TEST_FINISHED();
END_METHOD

METHOD PUBLIC Check_DATE_TO_TOD_TooHigh
VAR
	value : DATE := DatatypeLimits.DATE_MAX_VALUE;
	actual : TOD;
	converted : BOOL;
END_VAR
TEST('Check_DATE_TO_TOD_TooHigh');

// @TEST-RUN
converted := TryConvert_DATE_TO_Destination(value, actual);

// @TEST-ASSERT
AssertFalse(Condition := converted, Message := 'Did not report DATE to TOD conversion was prevented');

TEST_FINISHED();
END_METHOD

METHOD PUBLIC Check_DATE_TO_TOD_Max
VAR
	value : DATE := DatatypeLimits.MAX_VALUE_OF_DATE_WHICH_CAN_BE_HELD_IN_A_TOD;
	actual : TOD;
	converted : BOOL;
	equal : BOOL;
END_VAR
TEST('Check_DATE_TO_TOD_Max');

// @TEST-RUN
converted := TryConvert_DATE_TO_Destination(value, actual);
equal := actual = DATE_TO_TOD(value);

// @TEST-ASSERT
AssertTrue(Condition := equal, Message := 'Did not convert DATE to TOD correctly');
AssertTrue(Condition := converted, Message := 'Did not report DATE to TOD conversion was successful');

TEST_FINISHED();
END_METHOD

METHOD PUBLIC Check_DATE_TO_UDINT_Min
VAR
	value : DATE := DatatypeLimits.DATE_MIN_VALUE;
	actual : UDINT;
	converted : BOOL;
	equal : BOOL;
END_VAR
TEST('Check_DATE_TO_UDINT_Min');

// @TEST-RUN
converted := TryConvert_DATE_TO_Destination(value, actual);
equal := actual = DATE_TO_UDINT(value);

// @TEST-ASSERT
AssertTrue(Condition := equal, Message := 'Did not convert DATE to UDINT correctly');
AssertTrue(Condition := converted, Message := 'Did not report DATE to UDINT conversion was successful');

TEST_FINISHED();
END_METHOD

METHOD PUBLIC Check_DATE_TO_UDINT_Max
VAR
	value : DATE := DatatypeLimits.DATE_MAX_VALUE;
	actual : UDINT;
	converted : BOOL;
	equal : BOOL;
END_VAR
TEST('Check_DATE_TO_UDINT_Max');

// @TEST-RUN
converted := TryConvert_DATE_TO_Destination(value, actual);
equal := actual = DATE_TO_UDINT(value);

// @TEST-ASSERT
AssertTrue(Condition := equal, Message := 'Did not convert DATE to UDINT correctly');
AssertTrue(Condition := converted, Message := 'Did not report DATE to UDINT conversion was successful');

TEST_FINISHED();
END_METHOD

METHOD PUBLIC Check_DATE_TO_UINT_Min
VAR
	value : DATE := DatatypeLimits.DATE_MIN_VALUE;
	actual : UINT;
	converted : BOOL;
	equal : BOOL;
END_VAR
TEST('Check_DATE_TO_UINT_Min');

// @TEST-RUN
converted := TryConvert_DATE_TO_Destination(value, actual);
equal := actual = DATE_TO_UINT(value);

// @TEST-ASSERT
AssertTrue(Condition := equal, Message := 'Did not convert DATE to UINT correctly');
AssertTrue(Condition := converted, Message := 'Did not report DATE to UINT conversion was successful');

TEST_FINISHED();
END_METHOD

METHOD PUBLIC Check_DATE_TO_UINT_TooHigh
VAR
	value : DATE := DatatypeLimits.DATE_MAX_VALUE;
	actual : UINT;
	converted : BOOL;
END_VAR
TEST('Check_DATE_TO_UINT_TooHigh');

// @TEST-RUN
converted := TryConvert_DATE_TO_Destination(value, actual);

// @TEST-ASSERT
AssertFalse(Condition := converted, Message := 'Did not report DATE to UINT conversion was prevented');

TEST_FINISHED();
END_METHOD

METHOD PUBLIC Check_DATE_TO_UINT_Max
VAR
	value : DATE := DatatypeLimits.MAX_VALUE_OF_DATE_WHICH_CAN_BE_HELD_IN_A_UINT;
	actual : UINT;
	converted : BOOL;
	equal : BOOL;
END_VAR
TEST('Check_DATE_TO_UINT_Max');

// @TEST-RUN
converted := TryConvert_DATE_TO_Destination(value, actual);
equal := actual = DATE_TO_UINT(value);

// @TEST-ASSERT
AssertTrue(Condition := equal, Message := 'Did not convert DATE to UINT correctly');
AssertTrue(Condition := converted, Message := 'Did not report DATE to UINT conversion was successful');

TEST_FINISHED();
END_METHOD

METHOD PUBLIC Check_DATE_TO_ULINT_Min
VAR
	value : DATE := DatatypeLimits.DATE_MIN_VALUE;
	actual : ULINT;
	converted : BOOL;
	equal : BOOL;
END_VAR
TEST('Check_DATE_TO_ULINT_Min');

// @TEST-RUN
converted := TryConvert_DATE_TO_Destination(value, actual);
equal := actual = DATE_TO_ULINT(value);

// @TEST-ASSERT
AssertTrue(Condition := equal, Message := 'Did not convert DATE to ULINT correctly');
AssertTrue(Condition := converted, Message := 'Did not report DATE to ULINT conversion was successful');

TEST_FINISHED();
END_METHOD

METHOD PUBLIC Check_DATE_TO_ULINT_Max
VAR
	value : DATE := DatatypeLimits.DATE_MAX_VALUE;
	actual : ULINT;
	converted : BOOL;
	equal : BOOL;
END_VAR
TEST('Check_DATE_TO_ULINT_Max');

// @TEST-RUN
converted := TryConvert_DATE_TO_Destination(value, actual);
equal := actual = DATE_TO_ULINT(value);

// @TEST-ASSERT
AssertTrue(Condition := equal, Message := 'Did not convert DATE to ULINT correctly');
AssertTrue(Condition := converted, Message := 'Did not report DATE to ULINT conversion was successful');

TEST_FINISHED();
END_METHOD

METHOD PUBLIC Check_DATE_TO_USINT_Min
VAR
	value : DATE := DatatypeLimits.DATE_MIN_VALUE;
	actual : USINT;
	converted : BOOL;
	equal : BOOL;
END_VAR
TEST('Check_DATE_TO_USINT_Min');

// @TEST-RUN
converted := TryConvert_DATE_TO_Destination(value, actual);
equal := actual = DATE_TO_USINT(value);

// @TEST-ASSERT
AssertTrue(Condition := equal, Message := 'Did not convert DATE to USINT correctly');
AssertTrue(Condition := converted, Message := 'Did not report DATE to USINT conversion was successful');

TEST_FINISHED();
END_METHOD

METHOD PUBLIC Check_DATE_TO_USINT_TooHigh
VAR
	value : DATE := DatatypeLimits.DATE_MAX_VALUE;
	actual : USINT;
	converted : BOOL;
END_VAR
TEST('Check_DATE_TO_USINT_TooHigh');

// @TEST-RUN
converted := TryConvert_DATE_TO_Destination(value, actual);

// @TEST-ASSERT
AssertFalse(Condition := converted, Message := 'Did not report DATE to USINT conversion was prevented');

TEST_FINISHED();
END_METHOD

METHOD PUBLIC Check_DATE_TO_USINT_Max
VAR
	value : DATE := DatatypeLimits.MAX_VALUE_OF_DATE_WHICH_CAN_BE_HELD_IN_A_USINT;
	actual : USINT;
	converted : BOOL;
	equal : BOOL;
END_VAR
TEST('Check_DATE_TO_USINT_Max');

// @TEST-RUN
converted := TryConvert_DATE_TO_Destination(value, actual);
equal := actual = DATE_TO_USINT(value);

// @TEST-ASSERT
AssertTrue(Condition := equal, Message := 'Did not convert DATE to USINT correctly');
AssertTrue(Condition := converted, Message := 'Did not report DATE to USINT conversion was successful');

TEST_FINISHED();
END_METHOD

METHOD PUBLIC Check_DATE_TO_WORD_Min
VAR
	value : DATE := DatatypeLimits.DATE_MIN_VALUE;
	actual : WORD;
	converted : BOOL;
	equal : BOOL;
END_VAR
TEST('Check_DATE_TO_WORD_Min');

// @TEST-RUN
converted := TryConvert_DATE_TO_Destination(value, actual);
equal := actual = DATE_TO_WORD(value);

// @TEST-ASSERT
AssertTrue(Condition := equal, Message := 'Did not convert DATE to WORD correctly');
AssertTrue(Condition := converted, Message := 'Did not report DATE to WORD conversion was successful');

TEST_FINISHED();
END_METHOD

METHOD PUBLIC Check_DATE_TO_WORD_TooHigh
VAR
	value : DATE := DatatypeLimits.DATE_MAX_VALUE;
	actual : WORD;
	converted : BOOL;
END_VAR
TEST('Check_DATE_TO_WORD_TooHigh');

// @TEST-RUN
converted := TryConvert_DATE_TO_Destination(value, actual);

// @TEST-ASSERT
AssertFalse(Condition := converted, Message := 'Did not report DATE to WORD conversion was prevented');

TEST_FINISHED();
END_METHOD

METHOD PUBLIC Check_DATE_TO_WORD_Max
VAR
	value : DATE := DatatypeLimits.MAX_VALUE_OF_DATE_WHICH_CAN_BE_HELD_IN_A_WORD;
	actual : WORD;
	converted : BOOL;
	equal : BOOL;
END_VAR
TEST('Check_DATE_TO_WORD_Max');

// @TEST-RUN
converted := TryConvert_DATE_TO_Destination(value, actual);
equal := actual = DATE_TO_WORD(value);

// @TEST-ASSERT
AssertTrue(Condition := equal, Message := 'Did not convert DATE to WORD correctly');
AssertTrue(Condition := converted, Message := 'Did not report DATE to WORD conversion was successful');

TEST_FINISHED();
END_METHOD

END_FUNCTION_BLOCK

// ---- Tests/DT_TO_TestSuite.TcPOU
FUNCTION_BLOCK PUBLIC DT_TO_TestSuite EXTENDS TcUnit.FB_TestSuite
VAR
END_VAR

Check_DT_TO_BOOL_Max();
Check_DT_TO_BOOL_Min();
Check_DT_TO_BYTE_Max();
Check_DT_TO_BYTE_Min();
Check_DT_TO_BYTE_TooHigh();
Check_DT_TO_WORD_Max();
Check_DT_TO_WORD_Min();
Check_DT_TO_WORD_TooHigh();
Check_DT_TO_DWORD_Max();
Check_DT_TO_DWORD_Min();
Check_DT_TO_LWORD_Max();
Check_DT_TO_LWORD_Min();
Check_DT_TO_SINT_Max();
Check_DT_TO_SINT_Min();
Check_DT_TO_SINT_TooHigh();
Check_DT_TO_INT_Max();
Check_DT_TO_INT_Min();
Check_DT_TO_INT_TooHigh();
Check_DT_TO_DINT_Max();
Check_DT_TO_DINT_Min();
Check_DT_TO_DINT_TooHigh();
Check_DT_TO_LINT_Max();
Check_DT_TO_LINT_Min();
Check_DT_TO_USINT_Max();
Check_DT_TO_USINT_Min();
Check_DT_TO_USINT_TooHigh();
Check_DT_TO_UINT_Max();
Check_DT_TO_UINT_Min();
Check_DT_TO_UINT_TooHigh();
Check_DT_TO_UDINT_Max();
Check_DT_TO_UDINT_Min();
Check_DT_TO_ULINT_Max();
Check_DT_TO_ULINT_Min();
Check_DT_TO_REAL_Max();
Check_DT_TO_REAL_Min();
Check_DT_TO_LREAL_Max();
Check_DT_TO_LREAL_Min();
Check_DT_TO_TIME_Max();
Check_DT_TO_TIME_Min();
Check_DT_TO_TIME_TooHigh();
Check_DT_TO_TOD_Max();
Check_DT_TO_TOD_Min();
Check_DT_TO_TOD_TooHigh();
Check_DT_TO_DATE_Max();
Check_DT_TO_DATE_Min();
Check_DT_TO_DT_Max();
Check_DT_TO_DT_Min();
Check_DT_TO_STRING_Max();
Check_DT_TO_STRING_Min();

METHOD PUBLIC Check_DT_TO_BOOL_Min
VAR
	value : DT := DatatypeLimits.DT_MIN_VALUE;
	actual : BOOL;
	converted : BOOL;
	equal : BOOL;
END_VAR
TEST('Check_DT_TO_BOOL_Min');

// @TEST-RUN
converted := TryConvert_DT_TO_Destination(value, actual);
equal := actual = DT_TO_BOOL(value);

// @TEST-ASSERT
AssertTrue(Condition := equal, Message := 'Did not convert DT to BOOL correctly');
AssertTrue(Condition := converted, Message := 'Did not report DT to BOOL conversion was successful');

TEST_FINISHED();
END_METHOD

METHOD PUBLIC Check_DT_TO_BOOL_Max
VAR
	value : DT := DatatypeLimits.DT_MAX_VALUE;
	actual : BOOL;
	converted : BOOL;
	equal : BOOL;
END_VAR
TEST('Check_DT_TO_BOOL_Max');

// @TEST-RUN
converted := TryConvert_DT_TO_Destination(value, actual);
equal := actual = DT_TO_BOOL(value);

// @TEST-ASSERT
AssertTrue(Condition := equal, Message := 'Did not convert DT to BOOL correctly');
AssertTrue(Condition := converted, Message := 'Did not report DT to BOOL conversion was successful');

TEST_FINISHED();
END_METHOD

METHOD PUBLIC Check_DT_TO_BYTE_Min
VAR
	value : DT := DatatypeLimits.DT_MIN_VALUE;
	actual : BYTE;
	converted : BOOL;
	equal : BOOL;
END_VAR
TEST('Check_DT_TO_BYTE_Min');

// @TEST-RUN
converted := TryConvert_DT_TO_Destination(value, actual);
equal := actual = DT_TO_BYTE(value);

// @TEST-ASSERT
AssertTrue(Condition := equal, Message := 'Did not convert DT to BYTE correctly');
AssertTrue(Condition := converted, Message := 'Did not report DT to BYTE conversion was successful');

TEST_FINISHED();
END_METHOD

METHOD PUBLIC Check_DT_TO_BYTE_TooHigh
VAR
	value : DT := DatatypeLimits.DT_MAX_VALUE;
	actual : BYTE;
	converted : BOOL;
END_VAR
TEST('Check_DT_TO_BYTE_TooHigh');

// @TEST-RUN
converted := TryConvert_DT_TO_Destination(value, actual);

// @TEST-ASSERT
AssertFalse(Condition := converted, Message := 'Did not report DT to BYTE conversion was prevented');

TEST_FINISHED();
END_METHOD

METHOD PUBLIC Check_DT_TO_BYTE_Max
VAR
	value : DT := DatatypeLimits.MAX_VALUE_OF_DT_WHICH_CAN_BE_HELD_IN_A_BYTE;
	actual : BYTE;
	converted : BOOL;
	equal : BOOL;
END_VAR
TEST('Check_DT_TO_BYTE_Max');

// @TEST-RUN
converted := TryConvert_DT_TO_Destination(value, actual);
equal := actual = DT_TO_BYTE(value);

// @TEST-ASSERT
AssertTrue(Condition := equal, Message := 'Did not convert DT to BYTE correctly');
AssertTrue(Condition := converted, Message := 'Did not report DT to BYTE conversion was successful');

TEST_FINISHED();
END_METHOD

METHOD PUBLIC Check_DT_TO_DATE_Min
VAR
	value : DT := DatatypeLimits.DT_MIN_VALUE;
	actual : DATE;
	converted : BOOL;
	equal : BOOL;
END_VAR
TEST('Check_DT_TO_DATE_Min');

// @TEST-RUN
converted := TryConvert_DT_TO_Destination(value, actual);
equal := actual = DT_TO_DATE(value);

// @TEST-ASSERT
AssertTrue(Condition := equal, Message := 'Did not convert DT to DATE correctly');
AssertTrue(Condition := converted, Message := 'Did not report DT to DATE conversion was successful');

TEST_FINISHED();
END_METHOD

METHOD PUBLIC Check_DT_TO_DATE_Max
VAR
	value : DT := DatatypeLimits.DT_MAX_VALUE;
	actual : DATE;
	converted : BOOL;
	equal : BOOL;
END_VAR
TEST('Check_DT_TO_DATE_Max');

// @TEST-RUN
converted := TryConvert_DT_TO_Destination(value, actual);
equal := actual = DT_TO_DATE(value);

// @TEST-ASSERT
AssertTrue(Condition := equal, Message := 'Did not convert DT to DATE correctly');
AssertTrue(Condition := converted, Message := 'Did not report DT to DATE conversion was successful');

TEST_FINISHED();
END_METHOD

METHOD PUBLIC Check_DT_TO_DINT_Min
VAR
	value : DT := DatatypeLimits.DT_MIN_VALUE;
	actual : DINT;
	converted : BOOL;
	equal : BOOL;
END_VAR
TEST('Check_DT_TO_DINT_Min');

// @TEST-RUN
converted := TryConvert_DT_TO_Destination(value, actual);
equal := actual = DT_TO_DINT(value);

// @TEST-ASSERT
AssertTrue(Condition := equal, Message := 'Did not convert DT to DINT correctly');
AssertTrue(Condition := converted, Message := 'Did not report DT to DINT conversion was successful');

TEST_FINISHED();
END_METHOD

METHOD PUBLIC Check_DT_TO_DINT_TooHigh
VAR
	value : DT := DatatypeLimits.DT_MAX_VALUE;
	actual : DINT;
	converted : BOOL;
END_VAR
TEST('Check_DT_TO_DINT_TooHigh');

// @TEST-RUN
converted := TryConvert_DT_TO_Destination(value, actual);

// @TEST-ASSERT
AssertFalse(Condition := converted, Message := 'Did not report DT to DINT conversion was prevented');

TEST_FINISHED();
END_METHOD

METHOD PUBLIC Check_DT_TO_DINT_Max
VAR
	value : DT := DatatypeLimits.MAX_VALUE_OF_DT_WHICH_CAN_BE_HELD_IN_A_DINT;
	actual : DINT;
	converted : BOOL;
	equal : BOOL;
END_VAR
TEST('Check_DT_TO_DINT_Max');

// @TEST-RUN
converted := TryConvert_DT_TO_Destination(value, actual);
equal := actual = DT_TO_DINT(value);

// @TEST-ASSERT
AssertTrue(Condition := equal, Message := 'Did not convert DT to DINT correctly');
AssertTrue(Condition := converted, Message := 'Did not report DT to DINT conversion was successful');

TEST_FINISHED();
END_METHOD

METHOD PUBLIC Check_DT_TO_DT_Min
VAR
	value : DT := DatatypeLimits.DT_MIN_VALUE;
	actual : DT;
	converted : BOOL;
	equal : BOOL;
END_VAR
TEST('Check_DT_TO_DT_Min');

// @TEST-RUN
converted := TryConvert_DT_TO_Destination(value, actual);
equal := actual = value;

// @TEST-ASSERT
AssertTrue(Condition := equal, Message := 'Did not convert DT to DT correctly');
AssertTrue(Condition := converted, Message := 'Did not report DT to DT conversion was successful');

TEST_FINISHED();
END_METHOD

METHOD PUBLIC Check_DT_TO_DT_Max
VAR
	value : DT := DatatypeLimits.DT_MAX_VALUE;
	actual : DT;
	converted : BOOL;
	equal : BOOL;
END_VAR
TEST('Check_DT_TO_DT_Max');

// @TEST-RUN
converted := TryConvert_DT_TO_Destination(value, actual);
equal := actual = value;

// @TEST-ASSERT
AssertTrue(Condition := equal, Message := 'Did not convert DT to DT correctly');
AssertTrue(Condition := converted, Message := 'Did not report DT to DT conversion was successful');

TEST_FINISHED();
END_METHOD

METHOD PUBLIC Check_DT_TO_DWORD_Min
VAR
	value : DT := DatatypeLimits.DT_MIN_VALUE;
	actual : DWORD;
	converted : BOOL;
	equal : BOOL;
END_VAR
TEST('Check_DT_TO_DWORD_Min');

// @TEST-RUN
converted := TryConvert_DT_TO_Destination(value, actual);
equal := actual = DT_TO_DWORD(value);

// @TEST-ASSERT
AssertTrue(Condition := equal, Message := 'Did not convert DT to DWORD correctly');
AssertTrue(Condition := converted, Message := 'Did not report DT to DWORD conversion was successful');

TEST_FINISHED();
END_METHOD

METHOD PUBLIC Check_DT_TO_DWORD_Max
VAR
	value : DT := DatatypeLimits.DT_MAX_VALUE;
	actual : DWORD;
	converted : BOOL;
	equal : BOOL;
END_VAR
TEST('Check_DT_TO_DWORD_Max');

// @TEST-RUN
converted := TryConvert_DT_TO_Destination(value, actual);
equal := actual = DT_TO_DWORD(value);

// @TEST-ASSERT
AssertTrue(Condition := equal, Message := 'Did not convert DT to DWORD correctly');
AssertTrue(Condition := converted, Message := 'Did not report DT to DWORD conversion was successful');

TEST_FINISHED();
END_METHOD

METHOD PUBLIC Check_DT_TO_INT_Min
VAR
	value : DT := DatatypeLimits.DT_MIN_VALUE;
	actual : INT;
	converted : BOOL;
	equal : BOOL;
END_VAR
TEST('Check_DT_TO_INT_Min');

// @TEST-RUN
converted := TryConvert_DT_TO_Destination(value, actual);
equal := actual = DT_TO_INT(value);

// @TEST-ASSERT
AssertTrue(Condition := equal, Message := 'Did not convert DT to INT correctly');
AssertTrue(Condition := converted, Message := 'Did not report DT to INT conversion was successful');

TEST_FINISHED();
END_METHOD

METHOD PUBLIC Check_DT_TO_INT_TooHigh
VAR
	value : DT := DatatypeLimits.DT_MAX_VALUE;
	actual : INT;
	converted : BOOL;
END_VAR
TEST('Check_DT_TO_INT_TooHigh');

// @TEST-RUN
converted := TryConvert_DT_TO_Destination(value, actual);

// @TEST-ASSERT
AssertFalse(Condition := converted, Message := 'Did not report DT to INT conversion was prevented');

TEST_FINISHED();
END_METHOD

METHOD PUBLIC Check_DT_TO_INT_Max
VAR
	value : DT := DatatypeLimits.MAX_VALUE_OF_DT_WHICH_CAN_BE_HELD_IN_A_INT;
	actual : INT;
	converted : BOOL;
	equal : BOOL;
END_VAR
TEST('Check_DT_TO_INT_Max');

// @TEST-RUN
converted := TryConvert_DT_TO_Destination(value, actual);
equal := actual = DT_TO_INT(value);

// @TEST-ASSERT
AssertTrue(Condition := equal, Message := 'Did not convert DT to INT correctly');
AssertTrue(Condition := converted, Message := 'Did not report DT to INT conversion was successful');

TEST_FINISHED();
END_METHOD

METHOD PUBLIC Check_DT_TO_LINT_Min
VAR
	value : DT := DatatypeLimits.DT_MIN_VALUE;
	actual : LINT;
	converted : BOOL;
	equal : BOOL;
END_VAR
TEST('Check_DT_TO_LINT_Min');

// @TEST-RUN
converted := TryConvert_DT_TO_Destination(value, actual);
equal := actual = DT_TO_LINT(value);

// @TEST-ASSERT
AssertTrue(Condition := equal, Message := 'Did not convert DT to LINT correctly');
AssertTrue(Condition := converted, Message := 'Did not report DT to LINT conversion was successful');

TEST_FINISHED();
END_METHOD

METHOD PUBLIC Check_DT_TO_LINT_Max
VAR
	value : DT := DatatypeLimits.DT_MAX_VALUE;
	actual : LINT;
	converted : BOOL;
	equal : BOOL;
END_VAR
TEST('Check_DT_TO_LINT_Max');

// @TEST-RUN
converted := TryConvert_DT_TO_Destination(value, actual);
equal := actual = DT_TO_LINT(value);

// @TEST-ASSERT
AssertTrue(Condition := equal, Message := 'Did not convert DT to LINT correctly');
AssertTrue(Condition := converted, Message := 'Did not report DT to LINT conversion was successful');

TEST_FINISHED();
END_METHOD

METHOD PUBLIC Check_DT_TO_LREAL_Min
VAR
	value : DT := DatatypeLimits.DT_MIN_VALUE;
	actual : LREAL;
	converted : BOOL;
	equal : BOOL;
END_VAR
TEST('Check_DT_TO_LREAL_Min');

// @TEST-RUN
converted := TryConvert_DT_TO_Destination(value, actual);
equal := actual = DT_TO_LREAL(value);

// @TEST-ASSERT
AssertTrue(Condition := equal, Message := 'Did not convert DT to LREAL correctly');
AssertTrue(Condition := converted, Message := 'Did not report DT to LREAL conversion was successful');

TEST_FINISHED();
END_METHOD

METHOD PUBLIC Check_DT_TO_LREAL_Max
VAR
	value : DT := DatatypeLimits.DT_MAX_VALUE;
	actual : LREAL;
	converted : BOOL;
	equal : BOOL;
END_VAR
TEST('Check_DT_TO_LREAL_Max');

// @TEST-RUN
converted := TryConvert_DT_TO_Destination(value, actual);
equal := actual = DT_TO_LREAL(value);

// @TEST-ASSERT
AssertTrue(Condition := equal, Message := 'Did not convert DT to LREAL correctly');
AssertTrue(Condition := converted, Message := 'Did not report DT to LREAL conversion was successful');

TEST_FINISHED();
END_METHOD

METHOD PUBLIC Check_DT_TO_LWORD_Min
VAR
	value : DT := DatatypeLimits.DT_MIN_VALUE;
	actual : LWORD;
	converted : BOOL;
	equal : BOOL;
END_VAR
TEST('Check_DT_TO_LWORD_Min');

// @TEST-RUN
converted := TryConvert_DT_TO_Destination(value, actual);
equal := actual = DT_TO_LWORD(value);

// @TEST-ASSERT
AssertTrue(Condition := equal, Message := 'Did not convert DT to LWORD correctly');
AssertTrue(Condition := converted, Message := 'Did not report DT to LWORD conversion was successful');

TEST_FINISHED();
END_METHOD

METHOD PUBLIC Check_DT_TO_LWORD_Max
VAR
	value : DT := DatatypeLimits.DT_MAX_VALUE;
	actual : LWORD;
	converted : BOOL;
	equal : BOOL;
END_VAR
TEST('Check_DT_TO_LWORD_Max');

// @TEST-RUN
converted := TryConvert_DT_TO_Destination(value, actual);
equal := actual = DT_TO_LWORD(value);

// @TEST-ASSERT
AssertTrue(Condition := equal, Message := 'Did not convert DT to LWORD correctly');
AssertTrue(Condition := converted, Message := 'Did not report DT to LWORD conversion was successful');

TEST_FINISHED();
END_METHOD

METHOD PUBLIC Check_DT_TO_REAL_Min
VAR
	value : DT := DatatypeLimits.DT_MIN_VALUE;
	actual : REAL;
	converted : BOOL;
	equal : BOOL;
END_VAR
TEST('Check_DT_TO_REAL_Min');

// @TEST-RUN
converted := TryConvert_DT_TO_Destination(value, actual);
equal := actual = DT_TO_REAL(value);

// @TEST-ASSERT
AssertTrue(Condition := equal, Message := 'Did not convert DT to REAL correctly');
AssertTrue(Condition := converted, Message := 'Did not report DT to REAL conversion was successful');

TEST_FINISHED();
END_METHOD

METHOD PUBLIC Check_DT_TO_REAL_Max
VAR
	value : DT := DatatypeLimits.DT_MAX_VALUE;
	actual : REAL;
	converted : BOOL;
	equal : BOOL;
END_VAR
TEST('Check_DT_TO_REAL_Max');

// @TEST-RUN
converted := TryConvert_DT_TO_Destination(value, actual);
equal := actual = DT_TO_REAL(value);

// @TEST-ASSERT
AssertTrue(Condition := equal, Message := 'Did not convert DT to REAL correctly');
AssertTrue(Condition := converted, Message := 'Did not report DT to REAL conversion was successful');

TEST_FINISHED();
END_METHOD

METHOD PUBLIC Check_DT_TO_SINT_Min
VAR
	value : DT := DatatypeLimits.DT_MIN_VALUE;
	actual : SINT;
	converted : BOOL;
	equal : BOOL;
END_VAR
TEST('Check_DT_TO_SINT_Min');

// @TEST-RUN
converted := TryConvert_DT_TO_Destination(value, actual);
equal := actual = DT_TO_SINT(value);

// @TEST-ASSERT
AssertTrue(Condition := equal, Message := 'Did not convert DT to SINT correctly');
AssertTrue(Condition := converted, Message := 'Did not report DT to SINT conversion was successful');

TEST_FINISHED();
END_METHOD

METHOD PUBLIC Check_DT_TO_SINT_TooHigh
VAR
	value : DT := DatatypeLimits.DT_MAX_VALUE;
	actual : SINT;
	converted : BOOL;
END_VAR
TEST('Check_DT_TO_SINT_TooHigh');

// @TEST-RUN
converted := TryConvert_DT_TO_Destination(value, actual);

// @TEST-ASSERT
AssertFalse(Condition := converted, Message := 'Did not report DT to SINT conversion was prevented');

TEST_FINISHED();
END_METHOD

METHOD PUBLIC Check_DT_TO_SINT_Max
VAR
	value : DT := DatatypeLimits.MAX_VALUE_OF_DT_WHICH_CAN_BE_HELD_IN_A_SINT;
	actual : SINT;
	converted : BOOL;
	equal : BOOL;
END_VAR
TEST('Check_DT_TO_SINT_Max');

// @TEST-RUN
converted := TryConvert_DT_TO_Destination(value, actual);
equal := actual = DT_TO_SINT(value);

// @TEST-ASSERT
AssertTrue(Condition := equal, Message := 'Did not convert DT to SINT correctly');
AssertTrue(Condition := converted, Message := 'Did not report DT to SINT conversion was successful');

TEST_FINISHED();
END_METHOD

METHOD PUBLIC Check_DT_TO_STRING_Min
VAR
	value : DT := DatatypeLimits.DT_MIN_VALUE;
	actual : STRING;
	converted : BOOL;
	equal : BOOL;
END_VAR
TEST('Check_DT_TO_STRING_Min');

// @TEST-RUN
converted := TryConvert_DT_TO_Destination(value, actual);
equal := actual = DT_TO_STRING(value);

// @TEST-ASSERT
AssertTrue(Condition := equal, Message := 'Did not convert DT to STRING correctly');
AssertTrue(Condition := converted, Message := 'Did not report DT to STRING conversion was successful');

TEST_FINISHED();
END_METHOD

METHOD PUBLIC Check_DT_TO_STRING_Max
VAR
	value : DT := DatatypeLimits.DT_MAX_VALUE;
	actual : STRING;
	converted : BOOL;
	equal : BOOL;
END_VAR
TEST('Check_DT_TO_STRING_Max');

// @TEST-RUN
converted := TryConvert_DT_TO_Destination(value, actual);
equal := actual = DT_TO_STRING(value);

// @TEST-ASSERT
AssertTrue(Condition := equal, Message := 'Did not convert DT to STRING correctly');
AssertTrue(Condition := converted, Message := 'Did not report DT to STRING conversion was successful');

TEST_FINISHED();
END_METHOD

METHOD PUBLIC Check_DT_TO_TIME_Min
VAR
	value : DT := DatatypeLimits.DT_MIN_VALUE;
	actual : TIME;
	converted : BOOL;
	equal : BOOL;
END_VAR
TEST('Check_DT_TO_TIME_Min');

// @TEST-RUN
converted := TryConvert_DT_TO_Destination(value, actual);
equal := actual = DT_TO_TIME(value);

// @TEST-ASSERT
AssertTrue(Condition := equal, Message := 'Did not convert DT to TIME correctly');
AssertTrue(Condition := converted, Message := 'Did not report DT to TIME conversion was successful');

TEST_FINISHED();
END_METHOD

METHOD PUBLIC Check_DT_TO_TIME_TooHigh
VAR
	value : DT := DatatypeLimits.DT_MAX_VALUE;
	actual : TIME;
	converted : BOOL;
END_VAR
TEST('Check_DT_TO_TIME_TooHigh');

// @TEST-RUN
converted := TryConvert_DT_TO_Destination(value, actual);

// @TEST-ASSERT
AssertFalse(Condition := converted, Message := 'Did not report DT to TIME conversion was prevented');

TEST_FINISHED();
END_METHOD

METHOD PUBLIC Check_DT_TO_TIME_Max
VAR
	value : DT := DatatypeLimits.MAX_VALUE_OF_DT_WHICH_CAN_BE_HELD_IN_A_TIME;
	actual : TIME;
	converted : BOOL;
	equal : BOOL;
END_VAR
TEST('Check_DT_TO_TIME_Max');

// @TEST-RUN
converted := TryConvert_DT_TO_Destination(value, actual);
equal := actual = DT_TO_TIME(value);

// @TEST-ASSERT
AssertTrue(Condition := equal, Message := 'Did not convert DT to TIME correctly');
AssertTrue(Condition := converted, Message := 'Did not report DT to TIME conversion was successful');

TEST_FINISHED();
END_METHOD

METHOD PUBLIC Check_DT_TO_TOD_Min
VAR
	value : DT := DatatypeLimits.DT_MIN_VALUE;
	actual : TOD;
	converted : BOOL;
	equal : BOOL;
END_VAR
TEST('Check_DT_TO_TOD_Min');

// @TEST-RUN
converted := TryConvert_DT_TO_Destination(value, actual);
equal := actual = DT_TO_TOD(value);

// @TEST-ASSERT
AssertTrue(Condition := equal, Message := 'Did not convert DT to TOD correctly');
AssertTrue(Condition := converted, Message := 'Did not report DT to TOD conversion was successful');

TEST_FINISHED();
END_METHOD

METHOD PUBLIC Check_DT_TO_TOD_TooHigh
VAR
	value : DT := DatatypeLimits.DT_MAX_VALUE;
	actual : TOD;
	converted : BOOL;
END_VAR
TEST('Check_DT_TO_TOD_TooHigh');

// @TEST-RUN
converted := TryConvert_DT_TO_Destination(value, actual);

// @TEST-ASSERT
AssertFalse(Condition := converted, Message := 'Did not report DT to TOD conversion was prevented');

TEST_FINISHED();
END_METHOD

METHOD PUBLIC Check_DT_TO_TOD_Max
VAR
	value : DT := DatatypeLimits.MAX_VALUE_OF_DT_WHICH_CAN_BE_HELD_IN_A_TOD;
	actual : TOD;
	converted : BOOL;
	equal : BOOL;
END_VAR
TEST('Check_DT_TO_TOD_Max');

// @TEST-RUN
converted := TryConvert_DT_TO_Destination(value, actual);
equal := actual = DT_TO_TOD(value);

// @TEST-ASSERT
AssertTrue(Condition := equal, Message := 'Did not convert DT to TOD correctly');
AssertTrue(Condition := converted, Message := 'Did not report DT to TOD conversion was successful');

TEST_FINISHED();
END_METHOD

METHOD PUBLIC Check_DT_TO_UDINT_Min
VAR
	value : DT := DatatypeLimits.DT_MIN_VALUE;
	actual : UDINT;
	converted : BOOL;
	equal : BOOL;
END_VAR
TEST('Check_DT_TO_UDINT_Min');

// @TEST-RUN
converted := TryConvert_DT_TO_Destination(value, actual);
equal := actual = DT_TO_UDINT(value);

// @TEST-ASSERT
AssertTrue(Condition := equal, Message := 'Did not convert DT to UDINT correctly');
AssertTrue(Condition := converted, Message := 'Did not report DT to UDINT conversion was successful');

TEST_FINISHED();
END_METHOD

METHOD PUBLIC Check_DT_TO_UDINT_Max
VAR
	value : DT := DatatypeLimits.DT_MAX_VALUE;
	actual : UDINT;
	converted : BOOL;
	equal : BOOL;
END_VAR
TEST('Check_DT_TO_UDINT_Max');

// @TEST-RUN
converted := TryConvert_DT_TO_Destination(value, actual);
equal := actual = DT_TO_UDINT(value);

// @TEST-ASSERT
AssertTrue(Condition := equal, Message := 'Did not convert DT to UDINT correctly');
AssertTrue(Condition := converted, Message := 'Did not report DT to UDINT conversion was successful');

TEST_FINISHED();
END_METHOD

METHOD PUBLIC Check_DT_TO_UINT_Min
VAR
	value : DT := DatatypeLimits.DT_MIN_VALUE;
	actual : UINT;
	converted : BOOL;
	equal : BOOL;
END_VAR
TEST('Check_DT_TO_UINT_Min');

// @TEST-RUN
converted := TryConvert_DT_TO_Destination(value, actual);
equal := actual = DT_TO_UINT(value);

// @TEST-ASSERT
AssertTrue(Condition := equal, Message := 'Did not convert DT to UINT correctly');
AssertTrue(Condition := converted, Message := 'Did not report DT to UINT conversion was successful');

TEST_FINISHED();
END_METHOD

METHOD PUBLIC Check_DT_TO_UINT_TooHigh
VAR
	value : DT := DatatypeLimits.DT_MAX_VALUE;
	actual : UINT;
	converted : BOOL;
END_VAR
TEST('Check_DT_TO_UINT_TooHigh');

// @TEST-RUN
converted := TryConvert_DT_TO_Destination(value, actual);

// @TEST-ASSERT
AssertFalse(Condition := converted, Message := 'Did not report DT to UINT conversion was prevented');

TEST_FINISHED();
END_METHOD

METHOD PUBLIC Check_DT_TO_UINT_Max
VAR
	value : DT := DatatypeLimits.MAX_VALUE_OF_DT_WHICH_CAN_BE_HELD_IN_A_UINT;
	actual : UINT;
	converted : BOOL;
	equal : BOOL;
END_VAR
TEST('Check_DT_TO_UINT_Max');

// @TEST-RUN
converted := TryConvert_DT_TO_Destination(value, actual);
equal := actual = DT_TO_UINT(value);

// @TEST-ASSERT
AssertTrue(Condition := equal, Message := 'Did not convert DT to UINT correctly');
AssertTrue(Condition := converted, Message := 'Did not report DT to UINT conversion was successful');

TEST_FINISHED();
END_METHOD

METHOD PUBLIC Check_DT_TO_ULINT_Min
VAR
	value : DT := DatatypeLimits.DT_MIN_VALUE;
	actual : ULINT;
	converted : BOOL;
	equal : BOOL;
END_VAR
TEST('Check_DT_TO_ULINT_Min');

// @TEST-RUN
converted := TryConvert_DT_TO_Destination(value, actual);
equal := actual = DT_TO_ULINT(value);

// @TEST-ASSERT
AssertTrue(Condition := equal, Message := 'Did not convert DT to ULINT correctly');
AssertTrue(Condition := converted, Message := 'Did not report DT to ULINT conversion was successful');

TEST_FINISHED();
END_METHOD

METHOD PUBLIC Check_DT_TO_ULINT_Max
VAR
	value : DT := DatatypeLimits.DT_MAX_VALUE;
	actual : ULINT;
	converted : BOOL;
	equal : BOOL;
END_VAR
TEST('Check_DT_TO_ULINT_Max');

// @TEST-RUN
converted := TryConvert_DT_TO_Destination(value, actual);
equal := actual = DT_TO_ULINT(value);

// @TEST-ASSERT
AssertTrue(Condition := equal, Message := 'Did not convert DT to ULINT correctly');
AssertTrue(Condition := converted, Message := 'Did not report DT to ULINT conversion was successful');

TEST_FINISHED();
END_METHOD

METHOD PUBLIC Check_DT_TO_USINT_Min
VAR
	value : DT := DatatypeLimits.DT_MIN_VALUE;
	actual : USINT;
	converted : BOOL;
	equal : BOOL;
END_VAR
TEST('Check_DT_TO_USINT_Min');

// @TEST-RUN
converted := TryConvert_DT_TO_Destination(value, actual);
equal := actual = DT_TO_USINT(value);

// @TEST-ASSERT
AssertTrue(Condition := equal, Message := 'Did not convert DT to USINT correctly');
AssertTrue(Condition := converted, Message := 'Did not report DT to USINT conversion was successful');

TEST_FINISHED();
END_METHOD

METHOD PUBLIC Check_DT_TO_USINT_TooHigh
VAR
	value : DT := DatatypeLimits.DT_MAX_VALUE;
	actual : USINT;
	converted : BOOL;
END_VAR
TEST('Check_DT_TO_USINT_TooHigh');

// @TEST-RUN
converted := TryConvert_DT_TO_Destination(value, actual);

// @TEST-ASSERT
AssertFalse(Condition := converted, Message := 'Did not report DT to USINT conversion was prevented');

TEST_FINISHED();
END_METHOD

METHOD PUBLIC Check_DT_TO_USINT_Max
VAR
	value : DT := DatatypeLimits.MAX_VALUE_OF_DT_WHICH_CAN_BE_HELD_IN_A_USINT;
	actual : USINT;
	converted : BOOL;
	equal : BOOL;
END_VAR
TEST('Check_DT_TO_USINT_Max');

// @TEST-RUN
converted := TryConvert_DT_TO_Destination(value, actual);
equal := actual = DT_TO_USINT(value);

// @TEST-ASSERT
AssertTrue(Condition := equal, Message := 'Did not convert DT to USINT correctly');
AssertTrue(Condition := converted, Message := 'Did not report DT to USINT conversion was successful');

TEST_FINISHED();
END_METHOD

METHOD PUBLIC Check_DT_TO_WORD_Min
VAR
	value : DT := DatatypeLimits.DT_MIN_VALUE;
	actual : WORD;
	converted : BOOL;
	equal : BOOL;
END_VAR
TEST('Check_DT_TO_WORD_Min');

// @TEST-RUN
converted := TryConvert_DT_TO_Destination(value, actual);
equal := actual = DT_TO_WORD(value);

// @TEST-ASSERT
AssertTrue(Condition := equal, Message := 'Did not convert DT to WORD correctly');
AssertTrue(Condition := converted, Message := 'Did not report DT to WORD conversion was successful');

TEST_FINISHED();
END_METHOD

METHOD PUBLIC Check_DT_TO_WORD_TooHigh
VAR
	value : DT := DatatypeLimits.DT_MAX_VALUE;
	actual : WORD;
	converted : BOOL;
END_VAR
TEST('Check_DT_TO_WORD_TooHigh');

// @TEST-RUN
converted := TryConvert_DT_TO_Destination(value, actual);

// @TEST-ASSERT
AssertFalse(Condition := converted, Message := 'Did not report DT to WORD conversion was prevented');

TEST_FINISHED();
END_METHOD

METHOD PUBLIC Check_DT_TO_WORD_Max
VAR
	value : DT := DatatypeLimits.MAX_VALUE_OF_DT_WHICH_CAN_BE_HELD_IN_A_WORD;
	actual : WORD;
	converted : BOOL;
	equal : BOOL;
END_VAR
TEST('Check_DT_TO_WORD_Max');

// @TEST-RUN
converted := TryConvert_DT_TO_Destination(value, actual);
equal := actual = DT_TO_WORD(value);

// @TEST-ASSERT
AssertTrue(Condition := equal, Message := 'Did not convert DT to WORD correctly');
AssertTrue(Condition := converted, Message := 'Did not report DT to WORD conversion was successful');

TEST_FINISHED();
END_METHOD

END_FUNCTION_BLOCK

// ---- Tests/STRING_TO_TestSuite.TcPOU
FUNCTION_BLOCK PUBLIC STRING_TO_TestSuite EXTENDS TcUnit.FB_TestSuite
VAR
END_VAR

Check_STRING_TO_BOOL_Valid();
Check_STRING_TO_BYTE_Valid();
Check_STRING_TO_BYTE_Invalid();
Check_STRING_TO_WORD_Valid();
Check_STRING_TO_WORD_Invalid();
Check_STRING_TO_DWORD_Valid();
Check_STRING_TO_DWORD_Invalid();
Check_STRING_TO_LWORD_Valid();
Check_STRING_TO_LWORD_Invalid();
Check_STRING_TO_SINT_Valid();
Check_STRING_TO_SINT_Invalid();
Check_STRING_TO_INT_Valid();
Check_STRING_TO_INT_Invalid();
Check_STRING_TO_DINT_Valid();
Check_STRING_TO_DINT_Invalid();
Check_STRING_TO_LINT_Valid();
Check_STRING_TO_LINT_Invalid();
Check_STRING_TO_USINT_Valid();
Check_STRING_TO_USINT_Invalid();
Check_STRING_TO_UINT_Valid();
Check_STRING_TO_UINT_Invalid();
Check_STRING_TO_UDINT_Valid();
Check_STRING_TO_UDINT_Invalid();
Check_STRING_TO_ULINT_Valid();
Check_STRING_TO_ULINT_Invalid();
Check_STRING_TO_REAL_Valid();
Check_STRING_TO_REAL_Invalid();
Check_STRING_TO_LREAL_Valid();
Check_STRING_TO_LREAL_Invalid();
Check_STRING_TO_TIME_Valid();
Check_STRING_TO_TIME_Invalid();
Check_STRING_TO_TOD_Valid();
Check_STRING_TO_TOD_Invalid();
Check_STRING_TO_DATE_Valid();
Check_STRING_TO_DATE_Invalid();
Check_STRING_TO_DT_Valid();
Check_STRING_TO_DT_Invalid();
Check_STRING_TO_STRING_Valid();

METHOD PUBLIC Check_STRING_TO_BOOL_Valid
VAR
	value : STRING := BOOL_TO_STRING(DatatypeLimits.BOOL_MAX_VALUE);
	actual : BOOL;
	converted : BOOL;
	equal : BOOL;
END_VAR
TEST('Check_STRING_TO_BOOL_Valid');

// @TEST-RUN
converted := TryConvert_STRING_TO_Destination(value, actual);
equal := actual = STRING_TO_BOOL(value);

// @TEST-ASSERT
AssertTrue(Condition := equal, Message := 'Did not convert STRING to BOOL correctly');
AssertTrue(Condition := converted, Message := 'Did not report STRING to BOOL conversion was successful');

TEST_FINISHED();
END_METHOD

METHOD PUBLIC Check_STRING_TO_BYTE_Invalid
VAR
	value : STRING := 'hello';
	actual : BYTE;
	converted : BOOL;
END_VAR
TEST('Check_STRING_TO_BYTE_Invalid');

// @TEST-RUN
converted := TryConvert_STRING_TO_Destination(value, actual);

// @TEST-ASSERT
AssertFalse(Condition := converted, Message := 'Did not report STRING to BYTE conversion was prevented');

TEST_FINISHED();
END_METHOD

METHOD PUBLIC Check_STRING_TO_BYTE_Valid
VAR
	value : STRING := BYTE_TO_STRING(DatatypeLimits.BYTE_MAX_VALUE);
	actual : BYTE;
	converted : BOOL;
	equal : BOOL;
END_VAR
TEST('Check_STRING_TO_BYTE_Valid');

// @TEST-RUN
converted := TryConvert_STRING_TO_Destination(value, actual);
equal := actual = STRING_TO_BYTE(value);

// @TEST-ASSERT
AssertTrue(Condition := equal, Message := 'Did not convert STRING to BYTE correctly');
AssertTrue(Condition := converted, Message := 'Did not report STRING to BYTE conversion was successful');

TEST_FINISHED();
END_METHOD

METHOD PUBLIC Check_STRING_TO_DATE_Invalid
VAR
	value : STRING := 'hello';
	actual : DATE;
	converted : BOOL;
END_VAR
TEST('Check_STRING_TO_DATE_Invalid');

// @TEST-RUN
converted := TryConvert_STRING_TO_Destination(value, actual);

// @TEST-ASSERT
AssertFalse(Condition := converted, Message := 'Did not report STRING to DATE conversion was prevented');

TEST_FINISHED();
END_METHOD

METHOD PUBLIC Check_STRING_TO_DATE_Valid
VAR
	value : STRING := DATE_TO_STRING(DatatypeLimits.DATE_MAX_VALUE);
	actual : DATE;
	converted : BOOL;
	equal : BOOL;
END_VAR
TEST('Check_STRING_TO_DATE_Valid');

// @TEST-RUN
converted := TryConvert_STRING_TO_Destination(value, actual);
equal := actual = STRING_TO_DATE(value);

// @TEST-ASSERT
AssertTrue(Condition := equal, Message := 'Did not convert STRING to DATE correctly');
AssertTrue(Condition := converted, Message := 'Did not report STRING to DATE conversion was successful');

TEST_FINISHED();
END_METHOD

METHOD PUBLIC Check_STRING_TO_DINT_Invalid
VAR
	value : STRING := 'hello';
	actual : DINT;
	converted : BOOL;
END_VAR
TEST('Check_STRING_TO_DINT_Invalid');

// @TEST-RUN
converted := TryConvert_STRING_TO_Destination(value, actual);

// @TEST-ASSERT
AssertFalse(Condition := converted, Message := 'Did not report STRING to DINT conversion was prevented');

TEST_FINISHED();
END_METHOD

METHOD PUBLIC Check_STRING_TO_DINT_Valid
VAR
	value : STRING := DINT_TO_STRING(DatatypeLimits.DINT_MAX_VALUE);
	actual : DINT;
	converted : BOOL;
	equal : BOOL;
END_VAR
TEST('Check_STRING_TO_DINT_Valid');

// @TEST-RUN
converted := TryConvert_STRING_TO_Destination(value, actual);
equal := actual = STRING_TO_DINT(value);

// @TEST-ASSERT
AssertTrue(Condition := equal, Message := 'Did not convert STRING to DINT correctly');
AssertTrue(Condition := converted, Message := 'Did not report STRING to DINT conversion was successful');

TEST_FINISHED();
END_METHOD

METHOD PUBLIC Check_STRING_TO_DT_Invalid
VAR
	value : STRING := 'hello';
	actual : DT;
	converted : BOOL;
END_VAR
TEST('Check_STRING_TO_DT_Invalid');

// @TEST-RUN
converted := TryConvert_STRING_TO_Destination(value, actual);

// @TEST-ASSERT
AssertFalse(Condition := converted, Message := 'Did not report STRING to DT conversion was prevented');

TEST_FINISHED();
END_METHOD

METHOD PUBLIC Check_STRING_TO_DT_Valid
VAR
	value : STRING := DT_TO_STRING(DatatypeLimits.DT_MAX_VALUE);
	actual : DT;
	converted : BOOL;
	equal : BOOL;
END_VAR
TEST('Check_STRING_TO_DT_Valid');

// @TEST-RUN
converted := TryConvert_STRING_TO_Destination(value, actual);
equal := actual = STRING_TO_DT(value);

// @TEST-ASSERT
AssertTrue(Condition := equal, Message := 'Did not convert STRING to DT correctly');
AssertTrue(Condition := converted, Message := 'Did not report STRING to DT conversion was successful');

TEST_FINISHED();
END_METHOD

METHOD PUBLIC Check_STRING_TO_DWORD_Invalid
VAR
	value : STRING := 'hello';
	actual : DWORD;
	converted : BOOL;
END_VAR
TEST('Check_STRING_TO_DWORD_Invalid');

// @TEST-RUN
converted := TryConvert_STRING_TO_Destination(value, actual);

// @TEST-ASSERT
AssertFalse(Condition := converted, Message := 'Did not report STRING to DWORD conversion was prevented');

TEST_FINISHED();
END_METHOD

METHOD PUBLIC Check_STRING_TO_DWORD_Valid
VAR
	value : STRING := DWORD_TO_STRING(DatatypeLimits.DWORD_MAX_VALUE);
	actual : DWORD;
	converted : BOOL;
	equal : BOOL;
END_VAR
TEST('Check_STRING_TO_DWORD_Valid');

// @TEST-RUN
converted := TryConvert_STRING_TO_Destination(value, actual);
equal := actual = STRING_TO_DWORD(value);

// @TEST-ASSERT
AssertTrue(Condition := equal, Message := 'Did not convert STRING to DWORD correctly');
AssertTrue(Condition := converted, Message := 'Did not report STRING to DWORD conversion was successful');

TEST_FINISHED();
END_METHOD

METHOD PUBLIC Check_STRING_TO_INT_Invalid
VAR
	value : STRING := 'hello';
	actual : INT;
	converted : BOOL;
END_VAR
TEST('Check_STRING_TO_INT_Invalid');

// @TEST-RUN
converted := TryConvert_STRING_TO_Destination(value, actual);

// @TEST-ASSERT
AssertFalse(Condition := converted, Message := 'Did not report STRING to INT conversion was prevented');

TEST_FINISHED();
END_METHOD

METHOD PUBLIC Check_STRING_TO_INT_Valid
VAR
	value : STRING := INT_TO_STRING(DatatypeLimits.INT_MAX_VALUE);
	actual : INT;
	converted : BOOL;
	equal : BOOL;
END_VAR
TEST('Check_STRING_TO_INT_Valid');

// @TEST-RUN
converted := TryConvert_STRING_TO_Destination(value, actual);
equal := actual = STRING_TO_INT(value);

// @TEST-ASSERT
AssertTrue(Condition := equal, Message := 'Did not convert STRING to INT correctly');
AssertTrue(Condition := converted, Message := 'Did not report STRING to INT conversion was successful');

TEST_FINISHED();
END_METHOD

METHOD PUBLIC Check_STRING_TO_LINT_Invalid
VAR
	value : STRING := 'hello';
	actual : LINT;
	converted : BOOL;
END_VAR
TEST('Check_STRING_TO_LINT_Invalid');

// @TEST-RUN
converted := TryConvert_STRING_TO_Destination(value, actual);

// @TEST-ASSERT
AssertFalse(Condition := converted, Message := 'Did not report STRING to LINT conversion was prevented');

TEST_FINISHED();
END_METHOD

METHOD PUBLIC Check_STRING_TO_LINT_Valid
VAR
	value : STRING := LINT_TO_STRING(DatatypeLimits.LINT_MAX_VALUE);
	actual : LINT;
	converted : BOOL;
	equal : BOOL;
END_VAR
TEST('Check_STRING_TO_LINT_Valid');

// @TEST-RUN
converted := TryConvert_STRING_TO_Destination(value, actual);
equal := actual = STRING_TO_LINT(value);

// @TEST-ASSERT
AssertTrue(Condition := equal, Message := 'Did not convert STRING to LINT correctly');
AssertTrue(Condition := converted, Message := 'Did not report STRING to LINT conversion was successful');

TEST_FINISHED();
END_METHOD

METHOD PUBLIC Check_STRING_TO_LREAL_Invalid
VAR
	value : STRING := 'hello';
	actual : LREAL;
	converted : BOOL;
END_VAR
TEST('Check_STRING_TO_LREAL_Invalid');

// @TEST-RUN
converted := TryConvert_STRING_TO_Destination(value, actual);

// @TEST-ASSERT
AssertFalse(Condition := converted, Message := 'Did not report STRING to LREAL conversion was prevented');

TEST_FINISHED();
END_METHOD

METHOD PUBLIC Check_STRING_TO_LREAL_Valid
VAR
	value : STRING := LREAL_TO_STRING(DatatypeLimits.MAX_VALUE_OF_LREAL_WHICH_CAN_BE_HELD_IN_A_STRING);
	actual : LREAL;
	converted : BOOL;
	equal : BOOL;
END_VAR
TEST('Check_STRING_TO_LREAL_Valid');

// @TEST-RUN
converted := TryConvert_STRING_TO_Destination(value, actual);
equal := actual = STRING_TO_LREAL(value);

// @TEST-ASSERT
AssertTrue(Condition := equal, Message := 'Did not convert STRING to LREAL correctly');
AssertTrue(Condition := converted, Message := 'Did not report STRING to LREAL conversion was successful');

TEST_FINISHED();
END_METHOD

METHOD PUBLIC Check_STRING_TO_LWORD_Invalid
VAR
	value : STRING := 'hello';
	actual : LWORD;
	converted : BOOL;
END_VAR
TEST('Check_STRING_TO_LWORD_Invalid');

// @TEST-RUN
converted := TryConvert_STRING_TO_Destination(value, actual);

// @TEST-ASSERT
AssertFalse(Condition := converted, Message := 'Did not report STRING to LWORD conversion was prevented');

TEST_FINISHED();
END_METHOD

METHOD PUBLIC Check_STRING_TO_LWORD_Valid
VAR
	value : STRING := LWORD_TO_STRING(DatatypeLimits.LWORD_MAX_VALUE);
	actual : LWORD;
	converted : BOOL;
	equal : BOOL;
END_VAR
TEST('Check_STRING_TO_LWORD_Valid');

// @TEST-RUN
converted := TryConvert_STRING_TO_Destination(value, actual);
equal := actual = STRING_TO_LWORD(value);

// @TEST-ASSERT
AssertTrue(Condition := equal, Message := 'Did not convert STRING to LWORD correctly');
AssertTrue(Condition := converted, Message := 'Did not report STRING to LWORD conversion was successful');

TEST_FINISHED();
END_METHOD

METHOD PUBLIC Check_STRING_TO_REAL_Invalid
VAR
	value : STRING := 'hello';
	actual : REAL;
	converted : BOOL;
END_VAR
TEST('Check_STRING_TO_REAL_Invalid');

// @TEST-RUN
converted := TryConvert_STRING_TO_Destination(value, actual);

// @TEST-ASSERT
AssertFalse(Condition := converted, Message := 'Did not report STRING to REAL conversion was prevented');

TEST_FINISHED();
END_METHOD

METHOD PUBLIC Check_STRING_TO_REAL_Valid
VAR
	value : STRING := REAL_TO_STRING(DatatypeLimits.REAL_MAX_VALUE);
	actual : REAL;
	converted : BOOL;
	equal : BOOL;
END_VAR
TEST('Check_STRING_TO_REAL_Valid');

// @TEST-RUN
converted := TryConvert_STRING_TO_Destination(value, actual);
equal := actual = STRING_TO_REAL(value);

// @TEST-ASSERT
AssertTrue(Condition := equal, Message := 'Did not convert STRING to REAL correctly');
AssertTrue(Condition := converted, Message := 'Did not report STRING to REAL conversion was successful');

TEST_FINISHED();
END_METHOD

METHOD PUBLIC Check_STRING_TO_SINT_Invalid
VAR
	value : STRING := 'hello';
	actual : SINT;
	converted : BOOL;
END_VAR
TEST('Check_STRING_TO_SINT_Invalid');

// @TEST-RUN
converted := TryConvert_STRING_TO_Destination(value, actual);

// @TEST-ASSERT
AssertFalse(Condition := converted, Message := 'Did not report STRING to SINT conversion was prevented');

TEST_FINISHED();
END_METHOD

METHOD PUBLIC Check_STRING_TO_SINT_Valid
VAR
	value : STRING := SINT_TO_STRING(DatatypeLimits.SINT_MAX_VALUE);
	actual : SINT;
	converted : BOOL;
	equal : BOOL;
END_VAR
TEST('Check_STRING_TO_SINT_Valid');

// @TEST-RUN
converted := TryConvert_STRING_TO_Destination(value, actual);
equal := actual = STRING_TO_SINT(value);

// @TEST-ASSERT
AssertTrue(Condition := equal, Message := 'Did not convert STRING to SINT correctly');
AssertTrue(Condition := converted, Message := 'Did not report STRING to SINT conversion was successful');

TEST_FINISHED();
END_METHOD

METHOD PUBLIC Check_STRING_TO_STRING_Valid
VAR
	value : STRING := 'hello';
	actual : STRING;
	converted : BOOL;
	equal : BOOL;
END_VAR
TEST('Check_STRING_TO_STRING_Valid');

// @TEST-RUN
converted := TryConvert_STRING_TO_Destination(value, actual);
equal := actual = value;

// @TEST-ASSERT
AssertTrue(Condition := equal, Message := 'Did not convert STRING to STRING correctly');
AssertTrue(Condition := converted, Message := 'Did not report STRING to STRING conversion was successful');

TEST_FINISHED();
END_METHOD

METHOD PUBLIC Check_STRING_TO_TIME_Invalid
VAR
	value : STRING := 'hello';
	actual : TIME;
	converted : BOOL;
END_VAR
TEST('Check_STRING_TO_TIME_Invalid');

// @TEST-RUN
converted := TryConvert_STRING_TO_Destination(value, actual);

// @TEST-ASSERT
AssertFalse(Condition := converted, Message := 'Did not report STRING to TIME conversion was prevented');

TEST_FINISHED();
END_METHOD

METHOD PUBLIC Check_STRING_TO_TIME_Valid
VAR
	value : STRING := TIME_TO_STRING(DatatypeLimits.TIME_MAX_VALUE);
	actual : TIME;
	converted : BOOL;
	equal : BOOL;
END_VAR
TEST('Check_STRING_TO_TIME_Valid');

// @TEST-RUN
converted := TryConvert_STRING_TO_Destination(value, actual);
equal := actual = STRING_TO_TIME(value);

// @TEST-ASSERT
AssertTrue(Condition := equal, Message := 'Did not convert STRING to TIME correctly');
AssertTrue(Condition := converted, Message := 'Did not report STRING to TIME conversion was successful');

TEST_FINISHED();
END_METHOD

METHOD PUBLIC Check_STRING_TO_TOD_Invalid
VAR
	value : STRING := 'hello';
	actual : TOD;
	converted : BOOL;
END_VAR
TEST('Check_STRING_TO_TOD_Invalid');

// @TEST-RUN
converted := TryConvert_STRING_TO_Destination(value, actual);

// @TEST-ASSERT
AssertFalse(Condition := converted, Message := 'Did not report STRING to TOD conversion was prevented');

TEST_FINISHED();
END_METHOD

METHOD PUBLIC Check_STRING_TO_TOD_Valid
VAR
	value : STRING := TOD_TO_STRING(DatatypeLimits.TOD_MAX_VALUE);
	actual : TOD;
	converted : BOOL;
	equal : BOOL;
END_VAR
TEST('Check_STRING_TO_TOD_Valid');

// @TEST-RUN
converted := TryConvert_STRING_TO_Destination(value, actual);
equal := actual = STRING_TO_TOD(value);

// @TEST-ASSERT
AssertTrue(Condition := equal, Message := 'Did not convert STRING to TOD correctly');
AssertTrue(Condition := converted, Message := 'Did not report STRING to TOD conversion was successful');

TEST_FINISHED();
END_METHOD

METHOD PUBLIC Check_STRING_TO_UDINT_Invalid
VAR
	value : STRING := 'hello';
	actual : UDINT;
	converted : BOOL;
END_VAR
TEST('Check_STRING_TO_UDINT_Invalid');

// @TEST-RUN
converted := TryConvert_STRING_TO_Destination(value, actual);

// @TEST-ASSERT
AssertFalse(Condition := converted, Message := 'Did not report STRING to UDINT conversion was prevented');

TEST_FINISHED();
END_METHOD

METHOD PUBLIC Check_STRING_TO_UDINT_Valid
VAR
	value : STRING := UDINT_TO_STRING(DatatypeLimits.UDINT_MAX_VALUE);
	actual : UDINT;
	converted : BOOL;
	equal : BOOL;
END_VAR
TEST('Check_STRING_TO_UDINT_Valid');

// @TEST-RUN
converted := TryConvert_STRING_TO_Destination(value, actual);
equal := actual = STRING_TO_UDINT(value);

// @TEST-ASSERT
AssertTrue(Condition := equal, Message := 'Did not convert STRING to UDINT correctly');
AssertTrue(Condition := converted, Message := 'Did not report STRING to UDINT conversion was successful');

TEST_FINISHED();
END_METHOD

METHOD PUBLIC Check_STRING_TO_UINT_Invalid
VAR
	value : STRING := 'hello';
	actual : UINT;
	converted : BOOL;
END_VAR
TEST('Check_STRING_TO_UINT_Invalid');

// @TEST-RUN
converted := TryConvert_STRING_TO_Destination(value, actual);

// @TEST-ASSERT
AssertFalse(Condition := converted, Message := 'Did not report STRING to UINT conversion was prevented');

TEST_FINISHED();
END_METHOD

METHOD PUBLIC Check_STRING_TO_UINT_Valid
VAR
	value : STRING := UINT_TO_STRING(DatatypeLimits.UINT_MAX_VALUE);
	actual : UINT;
	converted : BOOL;
	equal : BOOL;
END_VAR
TEST('Check_STRING_TO_UINT_Valid');

// @TEST-RUN
converted := TryConvert_STRING_TO_Destination(value, actual);
equal := actual = STRING_TO_UINT(value);

// @TEST-ASSERT
AssertTrue(Condition := equal, Message := 'Did not convert STRING to UINT correctly');
AssertTrue(Condition := converted, Message := 'Did not report STRING to UINT conversion was successful');

TEST_FINISHED();
END_METHOD

METHOD PUBLIC Check_STRING_TO_ULINT_Invalid
VAR
	value : STRING := 'hello';
	actual : ULINT;
	converted : BOOL;
END_VAR
TEST('Check_STRING_TO_ULINT_Invalid');

// @TEST-RUN
converted := TryConvert_STRING_TO_Destination(value, actual);

// @TEST-ASSERT
AssertFalse(Condition := converted, Message := 'Did not report STRING to ULINT conversion was prevented');

TEST_FINISHED();
END_METHOD

METHOD PUBLIC Check_STRING_TO_ULINT_Valid
VAR
	value : STRING := ULINT_TO_STRING(DatatypeLimits.ULINT_MAX_VALUE);
	actual : ULINT;
	converted : BOOL;
	equal : BOOL;
END_VAR
TEST('Check_STRING_TO_ULINT_Valid');

// @TEST-RUN
converted := TryConvert_STRING_TO_Destination(value, actual);
equal := actual = STRING_TO_ULINT(value);

// @TEST-ASSERT
AssertTrue(Condition := equal, Message := 'Did not convert STRING to ULINT correctly');
AssertTrue(Condition := converted, Message := 'Did not report STRING to ULINT conversion was successful');

TEST_FINISHED();
END_METHOD

METHOD PUBLIC Check_STRING_TO_USINT_Invalid
VAR
	value : STRING := 'hello';
	actual : USINT;
	converted : BOOL;
END_VAR
TEST('Check_STRING_TO_USINT_Invalid');

// @TEST-RUN
converted := TryConvert_STRING_TO_Destination(value, actual);

// @TEST-ASSERT
AssertFalse(Condition := converted, Message := 'Did not report STRING to USINT conversion was prevented');

TEST_FINISHED();
END_METHOD

METHOD PUBLIC Check_STRING_TO_USINT_Valid
VAR
	value : STRING := USINT_TO_STRING(DatatypeLimits.USINT_MAX_VALUE);
	actual : USINT;
	converted : BOOL;
	equal : BOOL;
END_VAR
TEST('Check_STRING_TO_USINT_Valid');

// @TEST-RUN
converted := TryConvert_STRING_TO_Destination(value, actual);
equal := actual = STRING_TO_USINT(value);

// @TEST-ASSERT
AssertTrue(Condition := equal, Message := 'Did not convert STRING to USINT correctly');
AssertTrue(Condition := converted, Message := 'Did not report STRING to USINT conversion was successful');

TEST_FINISHED();
END_METHOD

METHOD PUBLIC Check_STRING_TO_WORD_Invalid
VAR
	value : STRING := 'hello';
	actual : WORD;
	converted : BOOL;
END_VAR
TEST('Check_STRING_TO_WORD_Invalid');

// @TEST-RUN
converted := TryConvert_STRING_TO_Destination(value, actual);

// @TEST-ASSERT
AssertFalse(Condition := converted, Message := 'Did not report STRING to WORD conversion was prevented');

TEST_FINISHED();
END_METHOD

METHOD PUBLIC Check_STRING_TO_WORD_Valid
VAR
	value : STRING := WORD_TO_STRING(DatatypeLimits.WORD_MAX_VALUE);
	actual : WORD;
	converted : BOOL;
	equal : BOOL;
END_VAR
TEST('Check_STRING_TO_WORD_Valid');

// @TEST-RUN
converted := TryConvert_STRING_TO_Destination(value, actual);
equal := actual = STRING_TO_WORD(value);

// @TEST-ASSERT
AssertTrue(Condition := equal, Message := 'Did not convert STRING to WORD correctly');
AssertTrue(Condition := converted, Message := 'Did not report STRING to WORD conversion was successful');

TEST_FINISHED();
END_METHOD

END_FUNCTION_BLOCK
